FUNCTION_BLOCK FB_SituarPale_SFC
VAR_INPUT
    // SFC-Flags
    SFCPause: BOOL;
    SFCReset: BOOL;
    
    // Indicadores de sincronizacion
    Ack: BOOL := TRUE;
    Execute: BOOL;
    
    // Parametros
    TpoPaleEntrada: TIME := T#400MS;
    
    // Entradas
    PalePresencia: BOOL;
    PaleCodigoBit0: BOOL;
    PaleCodigoBit1: BOOL;
    PaleCodigoBit2: BOOL;    
END_VAR
VAR_OUTPUT
    // Indicadores de sincronizacion
    Done: BOOL;
    Ready: BOOL;
    
    // Parametros
    PaleCodigo: BYTE;
    
    // Salidas
    CintaMotorActiva: BOOL;
END_VAR
VAR
END_VAR

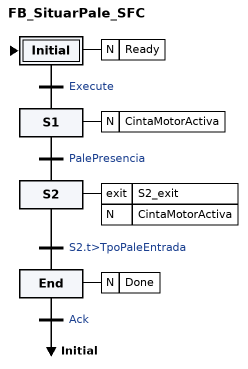
INITIAL_STEP Initial:
    Ready(N);
END_STEP
TRANSITION FROM Initial TO S1
    := Execute;
END_TRANSITION
STEP S1:
    CintaMotorActiva(N);
END_STEP
TRANSITION FROM S1 TO S2
    := PalePresencia;
END_TRANSITION
STEP S2:
    S2_exit(P0);  // exit action
    CintaMotorActiva(N);
END_STEP
TRANSITION FROM S2 TO End
    := S2.t>TpoPaleEntrada;
END_TRANSITION
STEP End:
    Done(N);
END_STEP
TRANSITION FROM End TO Initial
    := Ack;
END_TRANSITION

ACTION S2_exit:
PaleCodigo.0 := PaleCodigoBit0;
PaleCodigo.1 := PaleCodigoBit1;
PaleCodigo.2 := PaleCodigoBit2;
END_ACTION

END_FUNCTION_BLOCK

(* stored: Version 1.1.0.1, ProductVersion 3.1.4024.12
   POU FB_SituarPale_SFC: Id {874a499f-85d8-470a-bd97-def0802233cc}, SpecialFunc None
   Action S2_exit: Id {5e712388-189f-459b-a92a-f1a33cf515e1} *)
